Yaskawa INFORM job: MT_IN-MACHINE.JBI

/JOB
//NAME MT_IN-MACHINE
//POS
///NPOS 7,0,0,0,0,0
///TOOL 0
///POSTYPE PULSE
///PULSE
C00000=-60990,15190,81147,-73774,104817,21466
C00001=9470,155579,292637,-129341,95548,93543
C00002=5152,138415,271583,-125485,94027,-24675
C00003=485,131742,249882,-117145,94492,-117243
C00004=5152,138415,271583,-125485,94027,-24675
C00005=9470,155579,292637,-129341,95548,93543
C00006=-60990,15190,81147,-73774,104817,21466
//INST
///DATE 2023/10/12 17:18
///ATTR SC,RW
///GROUP1 RB1
NOP
MOVJ C00000 VJ=50.00
MOVJ C00001 VJ=50.00 PL=0
MOVJ C00002 VJ=50.00 PL=0
MOVJ C00003 VJ=50.00 PL=0
MOVJ C00004 VJ=50.00 PL=0
MOVJ C00005 VJ=50.00
MOVJ C00006 VJ=50.00
END
